{attribute 'qualified_only'}
VAR_GLOBAL
		EtherCAT_Master_BKCUCX : EtherCAT_Master_BKCUCX_11A6272B;
END_VAR

(* stored: Version 1.2.0.0, ProductVersion 3.1.4024.9
   GVL GVL_iXlinker: Id {2dc7ffd0-853b-451e-8f0f-317243e69d9b} *)
